ABB RobotStudio station: ABBRoboChallenge2022.rspag

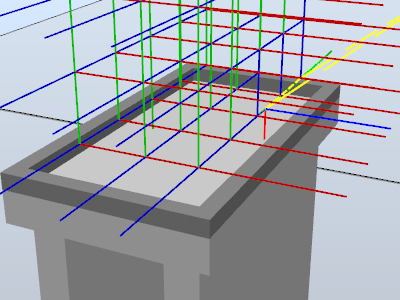
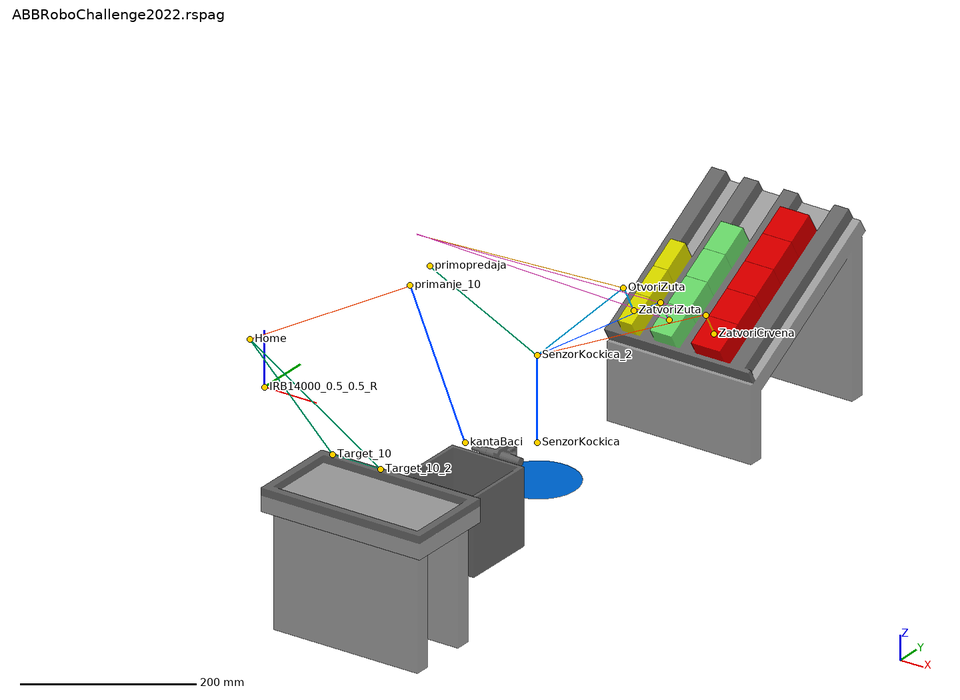
[picture v1: parts stored in the station drawn from their meshes, with robot base, taught points and paths (robot models come from the ABB library and are not in the file)]
--- station ---
Station Solution3 (saved by RobotStudio 22.3.10098.0)
Controller IRB14000, task T_ROB_L: task frame (RAPID world) sits at (0, 0, 100) mm in the station
Controller IRB14000, task T_ROB_R: task frame (RAPID world) sits at (0, 0, 100) mm in the station
Controller IRB14000
  mechanical unit ROB_R: IRB14000_0.5_0.5_R, 6 joints, base frame (0, 0, 0) mm
  mechanical unit ROB_R_7: IRB14000_0.5_0.5_R, 1 joints, base frame (0, 0, 0) mm
  mechanical unit ROB_L: IRB14000_0.5_0.5_L, 6 joints, base frame (0, 0, 0) mm
  mechanical unit ROB_L_7: IRB14000_0.5_0.5_L, 1 joints, base frame (0, 0, 0) mm
Layout (positions relative to the parent item):
  - IRB14000_0.5_0.5 [mechanism, from Robots\IRB14000_0.5_0.5__01.rslib] at (0, 0, 100) mm
  - IRB14000_0.5_0.5_R [mechanism, from Robots\IRB14000_0.5_0.5__01.rslib] at (0, 0, 100) mm; joint values [0.9031, -2.4871, -1.4074, 0.8318, -1.2822, 1.4209, -0.1871] (rad or m)
  - IRB14000_0.5_0.5_L [mechanism, from Robots\IRB14000_0.5_0.5__01.rslib] at (0, 0, 100) mm; joint values [-0.8577, -2.4871, 1.5284, 0.8395, 1.3372, 1.3689, -1.3488] (rad or m)
  - Smart_Gripper_Servo_One_Vacuum_Fingers [mechanism, from Tools\ABB_Smart_Gripper_Servo_One_Vacuum_Fingers.rslib] at (215.12, 134.2, 304.86) mm, rotated rx 113.54 ry -90 rz -23.54 deg; joint values [0] (rad or m)
  - Smart_Gripper_Servo_One_Vacuum_Camera_Fingers [mechanism, from Tools\ABB_Smart_Gripper_Servo_One_Vacuum_Camera_Fingers.rslib] at (228.58, -152.41, 307.36) mm, rotated rx 90 ry 0 rz -180 deg; joint values [0] (rad or m)
  - Senzor_Metala [part] at (250, 150, 15) mm, rotated rx 0 ry 0 rz 180 deg, size 65 x 32 x 27 mm
  - Mesto za testiranje [part] at (275, 150, 0) mm, size 100 x 99.5 x 0 mm
  - Rampa sa kutijama [graphiccomponentgroup]
    - Part_20 [part] at (374.5, 471.2, 184.6) mm, rotated rx 30 ry 0 rz 0 deg, size 40 x 40 x 40 mm
    - Part_1 [part] at (250, 320, 0) mm, size 200 x 20 x 100 mm
    - Part_2 [part] at (250, 520, 0) mm, size 200 x 20 x 200 mm
    - Part_3 [part], size 200 x 226.5 x 142.3 mm
    - Part_4 [part], size 200 x 14.3 x 19.8 mm
    - Part_5 [part], size 20 x 217.8 x 137.3 mm
    - Part_6 [part] at (45, 0, 0) mm, size 20 x 217.8 x 137.3 mm
    - Part_7 [part] at (100, 0, 0) mm, size 20 x 217.8 x 137.3 mm
    - Part_8 [part] at (170, 0, 0) mm, size 20 x 217.8 x 137.3 mm
    - Part_9 [part] at (292.5, 329.17, 102.6) mm, rotated rx 30 ry 0 rz 0 deg, size 20 x 40 x 40 mm
    - Part_10 [part] at (292.5, 364.68, 123.1) mm, rotated rx 30 ry 0 rz 0 deg, size 20 x 40 x 40 mm
    - Part_11 [part] at (292.5, 400.18, 143.6) mm, rotated rx 30 ry 0 rz 0 deg, size 20 x 40 x 40 mm
    - Part_12 [part] at (317.5, 329.17, 102.6) mm, rotated rx 30 ry 0 rz 0 deg, size 30 x 40 x 40 mm
    - Part_13 [part] at (317.5, 364.68, 123.1) mm, rotated rx 30 ry 0 rz 0 deg, size 30 x 40 x 40 mm
    - Part_14 [part] at (317.5, 400.18, 143.6) mm, rotated rx 30 ry 0 rz 0 deg, size 30 x 40 x 40 mm
    - Part_15 [part] at (374.5, 329.17, 102.6) mm, rotated rx 30 ry 0 rz 0 deg, size 40 x 40 x 40 mm
    - Part_16 [part] at (374.5, 364.68, 123.1) mm, rotated rx 30 ry 0 rz 0 deg, size 40 x 40 x 40 mm
    - Part_17 [part] at (374.5, 400.18, 143.6) mm, rotated rx 30 ry 0 rz 0 deg, size 40 x 40 x 40 mm
    - Part_18 [part] at (317.5, 435.69, 164.1) mm, rotated rx 30 ry 0 rz 0 deg, size 30 x 40 x 40 mm
    - Part_19 [part] at (374.5, 435.69, 164.1) mm, rotated rx 30 ry 0 rz 0 deg, size 40 x 40 x 40 mm
  - Paleta [graphiccomponentgroup]
    - Part_31 [part] at (450, -340, 170) mm, size 10 x 100 x 10 mm
    - Part_21 [part] at (250, -340, 0) mm, size 200 x 20 x 150 mm
    - Part_22 [part] at (250, -260, 0) mm, size 200 x 20 x 150 mm
    - Part_25 [part] at (240, -350, 170) mm, size 220 x 10 x 10 mm
    - Part_26 [part] at (240, -240, 170) mm, size 220 x 10 x 10 mm
    - Part_27 [part] at (240, -350, 150) mm, size 220 x 120 x 20 mm
    - Part_28 [part] at (240, -340, 170) mm, size 10 x 100 x 10 mm
  - Mesto za odlaganje [part], size 100 x 100 x 100 mm
Attachment: Smart_Gripper_Servo_One_Vacuum_Fingers is attached to IRB14000_0.5_0.5_L / Link7
Attachment: Smart_Gripper_Servo_One_Vacuum_Camera_Fingers is attached to IRB14000_0.5_0.5_R / Link7
Attachment: Part_8 is attached to Part_7
Attachment: Part_7 is attached to Part_6
Attachment: Part_6 is attached to Part_5
Attachment: Part_5 is attached to Part_4
Attachment: Part_4 is attached to Part_3
Attachment: Part_3 is attached to Part_2
Attachment: Part_2 is attached to Part_1
Attachment: Part_9 is attached to Part_4
Attachment: Part_10 is attached to Part_4
Attachment: Part_11 is attached to Part_4
Attachment: Part_12 is attached to Part_4
Attachment: Part_13 is attached to Part_4
Attachment: Part_14 is attached to Part_4
Attachment: Part_15 is attached to Part_4
Attachment: Part_16 is attached to Part_4
Attachment: Part_17 is attached to Part_4
Attachment: Part_18 is attached to Part_4
Attachment: Part_19 is attached to Part_4
Attachment: Part_20 is attached to Part_4
Attachment: Part_31 is attached to Part_28
Attachment: Part_28 is attached to Part_26
Attachment: Part_26 is attached to Part_25
Attachment: Part_25 is attached to Part_27
Attachment: Part_27 is attached to Part_22
Attachment: Part_22 is attached to Part_21
Targets, tools, work objects and paths stored in the station and not in the controller backup, written as RAPID:
! task T_ROB_L
MODULE Module1
  CONST robtarget SenzorKockica_2_4:=[[0,0,-0.911663764],[0,-0.707106781,0.707106781,0],[-1,0,1,5],[103.674755702,9E+09,9E+09,9E+09,9E+09,9E+09]];
  CONST robtarget SenzorKockica_4:=[[0,0,128.036682994],[0,0.707106781,0.707106781,0],[-1,0,1,5],[103.674755702,9E+09,9E+09,9E+09,9E+09,9E+09]];
ENDMODULE


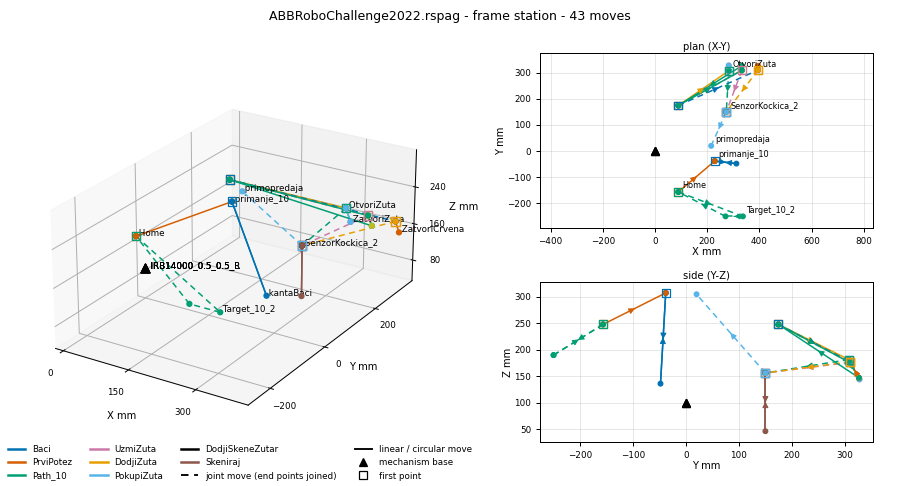
[picture p0: tool path of ABBRoboChallenge2022.rspag in frame station, 43 of 43 moves have a stored position in this frame; points joined in program order, loops and branches not executed]
--- Backups/IRB14000/RAPID/TASK1/PROGMOD/CalibData.mod ---
MODULE CalibData
    PERS tooldata Servo:=[TRUE,[[0,0,114.2],[1,0,0,0]],[0.24,[8.2,12.5,48.1],[1,0,0,0],0.00022,0.00024,0.00009]];
    PERS tooldata VaccumOne:=[TRUE,[[63.5,18.5,37.5],[0.707106781,0,0.707106781,0]],[0.24,[8.2,12.5,48.1],[1,0,0,0],0.00022,0.00024,0.00009]];
    PERS tooldata Camera:=[TRUE,[[-7.3,28.3,35.1],[0.5,-0.5,0.5,0.5]],[0.24,[8.2,12.5,48.1],[1,0,0,0],0.00022,0.00024,0.00009]];
    PERS wobjdata Workobject_2:=[FALSE,TRUE,"",[[311.493,-47.839,34.371],[1,0,0,0]],[[0,0,0],[1,0,0,0]]];
   PERS wobjdata Workobject_3:=[FALSE,TRUE,"",[[270,-250,90],[0.5,0.5,0.5,0.5]],[[0,0,0],[0.707106781,-0.707106781,0,0]]];
    PERS wobjdata Workobject_4:=[FALSE,TRUE,"",[[310,-250,90],[0.5,0.5,0.5,0.5]],[[0,0,0],[0.707106781,-0.707106781,0,0]]];
    PERS wobjdata Workobject_5:=[FALSE,TRUE,"",[[350,-250,90],[0.5,0.5,0.5,0.5]],[[0,0,0],[0.707106781,-0.707106781,0,0]]];
    PERS wobjdata Workobject_6:=[FALSE,TRUE,"",[[390,-250,90],[0.5,0.5,0.5,0.5]],[[0,0,0],[1,0,0,0]]];
    PERS wobjdata Workobject_7:=[FALSE,TRUE,"",[[430,-250,90],[0.5,0.5,0.5,0.5]],[[0,0,0],[1,0,0,0]]];
    PERS wobjdata Workobject_8:=[FALSE,TRUE,"",[[430,-320,90],[0.5,0.5,0.5,0.5]],[[0,0,0],[1,0,0,0]]];
    PERS wobjdata Workobject_9:=[FALSE,TRUE,"",[[390,-320,90],[0.5,0.5,0.5,0.5]],[[0,0,0],[1,0,0,0]]];
    PERS wobjdata Workobject_10:=[FALSE,TRUE,"",[[390,-280,90],[0.5,0.5,0.5,0.5]],[[0,0,0],[1,0,0,0]]];
    PERS wobjdata Workobject_11:=[FALSE,TRUE,"",[[430,-280,90],[0.5,0.5,0.5,0.5]],[[0,0,0],[1,0,0,0]]];
    PERS wobjdata Workobject_12:=[FALSE,TRUE,"",[[270,-320,90],[0.5,0.5,0.5,0.5]],[[0,0,0],[1,0,0,0]]];
    PERS wobjdata Workobject_13:=[FALSE,TRUE,"",[[270,-280,90],[0.5,0.5,0.5,0.5]],[[0,0,0],[1,0,0,0]]];
    PERS wobjdata Workobject_14:=[FALSE,TRUE,"",[[310,-320,90],[0.5,0.5,0.5,0.5]],[[0,0,0],[1,0,0,0]]];
    PERS wobjdata Workobject_15:=[FALSE,TRUE,"",[[310,-280,90],[0.5,0.5,0.5,0.5]],[[0,0,0],[1,0,0,0]]];
    PERS wobjdata Workobject_16:=[FALSE,TRUE,"",[[350,-280,90],[0.5,0.5,0.5,0.5]],[[0,0,0],[1,0,0,0]]];
    PERS wobjdata Workobject_17:=[FALSE,TRUE,"",[[350,-320,90],[0.5,0.5,0.5,0.5]],[[0,0,0],[0,1,0,0]]];
    PERS wobjdata Workobject_21:=[FALSE,TRUE,"",[[430,-320,130],[0.5,0.5,0.5,0.5]],[[0,0,0],[1,0,0,0]]];
    PERS wobjdata Workobject_22:=[FALSE,TRUE,"",[[390,-320,130],[0.5,0.5,0.5,0.5]],[[0,0,0],[1,0,0,0]]];
    PERS wobjdata Workobject_23:=[FALSE,TRUE,"",[[350,-320,130],[0.5,0.5,0.5,0.5]],[[0,0,0],[1,0,0,0]]];
    PERS wobjdata Workobject_24:=[FALSE,TRUE,"",[[310,-320,130],[0.5,0.5,0.5,0.5]],[[0,0,0],[1,0,0,0]]];
    PERS wobjdata Workobject_25:=[FALSE,TRUE,"",[[270,-320,130],[0.5,0.5,0.5,0.5]],[[0,0,0],[1,0,0,0]]];
    PERS wobjdata Workobject_26:=[FALSE,TRUE,"",[[270,-280,130],[0.5,0.5,0.5,0.5]],[[0,0,0],[1,0,0,0]]];
    PERS wobjdata Workobject_27:=[FALSE,TRUE,"",[[310,-280,130],[0.5,0.5,0.5,0.5]],[[0,0,0],[1,0,0,0]]];
    PERS wobjdata Workobject_28:=[FALSE,TRUE,"",[[350,-280,130],[0.5,0.5,0.5,0.5]],[[0,0,0],[1,0,0,0]]];
    PERS wobjdata Workobject_29:=[FALSE,TRUE,"",[[390,-280,130],[0.5,0.5,0.5,0.5]],[[0,0,0],[1,0,0,0]]];
    PERS wobjdata Workobject_30:=[FALSE,TRUE,"",[[430,-280,130],[0.5,0.5,0.5,0.5]],[[0,0,0],[1,0,0,0]]];
    PERS wobjdata Workobject_31:=[FALSE,TRUE,"",[[270,-250,130],[0.5,0.5,0.5,0.5]],[[0,0,0],[1,0,0,0]]];
    PERS wobjdata Workobject_32:=[FALSE,TRUE,"",[[310,-250,130],[0.5,0.5,0.5,0.5]],[[0,0,0],[1,0,0,0]]];
    PERS wobjdata Workobject_33:=[FALSE,TRUE,"",[[350,-250,130],[0.5,0.5,0.5,0.5]],[[0,0,0],[1,0,0,0]]];
    PERS wobjdata Workobject_34:=[FALSE,TRUE,"",[[390,-250,130],[0.5,0.5,0.5,0.5]],[[0,0,0],[1,0,0,0]]];
    PERS wobjdata Workobject_35:=[FALSE,TRUE,"",[[430,-250,130],[0.5,0.5,0.5,0.5]],[[0,0,0],[1,0,0,0]]];
    PERS wobjdata Workobject_36:=[FALSE,TRUE,"",[[430,-320,170],[0.5,0.5,0.5,0.5]],[[0,0,0],[1,0,0,0]]];
    PERS wobjdata Workobject_37:=[FALSE,TRUE,"",[[270,-320,170],[0.5,0.5,0.5,0.5]],[[0,0,0],[1,0,0,0]]];
    PERS wobjdata Workobject_38:=[FALSE,TRUE,"",[[270,-280,170],[0.5,0.5,0.5,0.5]],[[0,0,0],[1,0,0,0]]];
    PERS wobjdata Workobject_39:=[FALSE,TRUE,"",[[310,-320,170],[0.5,0.5,0.5,0.5]],[[0,0,0],[1,0,0,0]]];
    PERS wobjdata Workobject_40:=[FALSE,TRUE,"",[[310,-280,170],[0.5,0.5,0.5,0.5]],[[0,0,0],[1,0,0,0]]];
    PERS wobjdata Workobject_41:=[FALSE,TRUE,"",[[270,-250,170],[0.5,0.5,0.5,0.5]],[[0,0,0],[1,0,0,0]]];
    PERS wobjdata Workobject_42:=[FALSE,TRUE,"",[[310,-250,170],[0.5,0.5,0.5,0.5]],[[0,0,0],[1,0,0,0]]];
    PERS wobjdata Workobject_43:=[FALSE,TRUE,"",[[350,-320,170],[0.5,0.5,0.5,0.5]],[[0,0,0],[1,0,0,0]]];
    PERS wobjdata Workobject_44:=[FALSE,TRUE,"",[[350,-280,170],[0.5,0.5,0.5,0.5]],[[0,0,0],[1,0,0,0]]];
    PERS wobjdata Workobject_45:=[FALSE,TRUE,"",[[350,-250,170],[0.5,0.5,0.5,0.5]],[[0,0,0],[1,0,0,0]]];
    PERS wobjdata Workobject_46:=[FALSE,TRUE,"",[[390,-320,170],[0.5,0.5,0.5,0.5]],[[0,0,0],[1,0,0,0]]];
    PERS wobjdata Workobject_47:=[FALSE,TRUE,"",[[390,-280,170],[0.5,0.5,0.5,0.5]],[[0,0,0],[1,0,0,0]]];
    PERS wobjdata Workobject_48:=[FALSE,TRUE,"",[[430,-250,170],[0.5,0.5,0.5,0.5]],[[0,0,0],[1,0,0,0]]];
    PERS wobjdata Workobject_49:=[FALSE,TRUE,"",[[390,-250,170],[0.5,0.5,0.5,0.5]],[[0,0,0],[1,0,0,0]]];
    PERS wobjdata Workobject_50:=[FALSE,TRUE,"",[[430,-280,170],[0.5,0.5,0.5,0.5]],[[0,0,0],[1,0,0,0]]];
    PERS wobjdata Workobject_51:=[FALSE,TRUE,"",[[265,-20,190],[1,0,0,0]],[[0,0,0],[1,0,0,0]]];
    PERS wobjdata Kanta:=[FALSE,TRUE,"",[[311.493,-47.839,34.371],[0,1,0,0]],[[0,0,0],[1,0,0,0]]];
    PERS wobjdata Primanje:=[FALSE,TRUE,"",[[265,-20,190],[1,0,0,0]],[[0,0,0],[1,0,0,0]]];
    PERS wobjdata Workobject_1:=[FALSE,TRUE,"",[[273,150,-53.701],[1,0,0,0]],[[0,0,0],[1,0,0,0]]];
    PERS wobjdata KockicaZ:=[FALSE,TRUE,"",[[282.5,326.49,47.239],[0.969411434,0.245441382,0,0]],[[0,0,0],[1,0,0,0]]];
    PERS wobjdata Workobject_19:=[FALSE,TRUE,"",[[332.5,326.491,47.241],[1,0,0,0]],[[0,0,0],[1,0,0,0]]];
    PERS wobjdata Workobject_20:=[FALSE,TRUE,"",[[394.5,326.491,47.241],[0.608400247,-0.360345861,0.608400247,-0.360345861]],[[0,0,0],[1,0,0,0]]];
    PERS wobjdata Workobject_53:=[FALSE,TRUE,"",[[265,-26.752845654,190],[0.5,0.5,0.5,0.5]],[[0,0,0],[1,0,0,0]]];
ENDMODULE

--- Backups/IRB14000/RAPID/TASK1/PROGMOD/Module1.mod ---
MODULE Module1
        CONST robtarget primanje_10:=[[-36.418450574,-18.209391177,17.355412881],[0,0,0.707106781,0.707106781],[1,-1,0,4],[-101.964427132,9E+09,9E+09,9E+09,9E+09,9E+09]];
    CONST robtarget kanta_10:=[[0,0,0],[1,0,0,0],[-1,0,1,1],[-111.964425004,9E+09,9E+09,9E+09,9E+09,9E+09]];
    CONST robtarget Home:=[[89.387946422,-156.622117956,147.913470217],[0.066010726,-0.842420918,-0.111214912,-0.523068661],[0,0,0,4],[-101.964427132,9E+09,9E+09,9E+09,9E+09,9E+09]];
    CONST robtarget primopredaja_2:=[[0,0,0],[0.5,0.5,-0.5,0.5],[1,0,2,1],[103.674760418,9E+09,9E+09,9E+09,9E+09,9E+09]];
    CONST robtarget primanje_10_2:=[[0.267352692,0.235735351,-1.691583869],[0,0,0,1],[1,-1,0,4],[-101.964427132,9E+09,9E+09,9E+09,9E+09,9E+09]];
    CONST robtarget kantaBaci:=[[0.267352692,0.235735351,-1.691583869],[0,0,0,1],[1,-1,0,4],[-101.964427132,9E+09,9E+09,9E+09,9E+09,9E+09]];
    CONST robtarget Target_10:=[[0,0,0],[1,0,0,0],[1,0,-1,5],[-101.964427132,9E+09,9E+09,9E+09,9E+09,9E+09]];
    CONST robtarget Target_10_2:=[[0,-66.608628748,0],[0.707106781,0,0.707106781,0],[1,0,-1,5],[-101.964427132,9E+09,9E+09,9E+09,9E+09,9E+09]];
    CONST robtarget Target_20:=[[0,0,0],[1,0,0,0],[0,0,0,0],[-101.964417119,9E+09,9E+09,9E+09,9E+09,9E+09]];
    PROC main()
        Path_10;
    ENDPROC
    PROC Baci()
        MoveL primanje_10,v1000,z100,Servo\WObj:=Primanje;
        MoveL kantaBaci,v1000,z100,Servo\WObj:=Kanta;
        MoveL primanje_10,v1000,z100,Servo\WObj:=Primanje;
    ENDPROC
    PROC PrviPotez()
        MoveL Home,v1000,z100,Servo\WObj:=wobj0;
        MoveL primanje_10,v1000,z100,Servo\WObj:=Primanje;
    ENDPROC
    PROC Path_10()
        MoveL Home,v1000,z100,Servo\WObj:=wobj0;
        MoveJ Target_10_2,v1000,z100,Servo\WObj:=Workobject_3;
        MoveJ Target_10,v1000,z100,Servo\WObj:=Workobject_3;
        MoveJ Home,v1000,z100,Servo\WObj:=wobj0;
    ENDPROC
ENDMODULE

--- Backups/IRB14000/RAPID/TASK2/PROGMOD/CalibData.mod ---
MODULE CalibData
    PERS tooldata Servo:=[TRUE,[[0,0,114.2],[1,0,0,0]],[0.226,[8.9,12.3,48.7],[1,0,0,0],0.00021,0.00024,0.00009]];
    PERS tooldata VaccumOne:=[TRUE,[[63.5,18.5,37.5],[0.707106781,0,0.707106781,0]],[0.226,[8.9,12.3,48.7],[1,0,0,0],0.00021,0.00024,0.00009]];
    PERS wobjdata Workobject_1:=[FALSE,TRUE,"",[[273,150,-53.701],[1,0,0,0]],[[0,0,0],[1,0,0,0]]];
    PERS wobjdata KockicaZ:=[FALSE,TRUE,"",[[282.5,326.49,47.239],[0.969411434,0.245441382,0,0]],[[0,0,0],[1,0,0,0]]];
    PERS wobjdata Workobject_19:=[FALSE,TRUE,"",[[332.5,326.491,47.241],[1,0,0,0]],[[0,0,0],[1,0,0,0]]];
    PERS wobjdata Workobject_20:=[FALSE,TRUE,"",[[394.5,326.491,47.241],[0.248054386,-0.968746108,0,0]],[[0,0,0],[1,0,0,0]]];
    PERS wobjdata Workobject_51:=[FALSE,TRUE,"",[[265,-20,190],[1,0,0,0]],[[0,0,0],[1,0,0,0]]];
    PERS wobjdata Workobject_53:=[FALSE,TRUE,"",[[265,20,190],[1,0,0,0]],[[0,0,0],[1,0,0,0]]];
ENDMODULE

--- Backups/IRB14000/RAPID/TASK2/PROGMOD/Module1.mod ---
MODULE Module1
    CONST robtarget Home:=[[89.388081176,174.575150508,147.913525533],[0.06601065,0.842420935,-0.111215019,0.52306862],[0,0,0,4],[101.964427489,9E+09,9E+09,9E+09,9E+09,9E+09]];
    CONST robtarget OtvoriZuta:=[[0,-0.475935817,39.28134243],[-0.000001405,1,0,0],[-1,-2,2,4],[101.964427132,9E+09,9E+09,9E+09,9E+09,9E+09]];
    CONST robtarget ZatvoriZuta:=[[0,-0.476055148,-3.185077172],[-0.000001405,1,0,0],[-1,-2,2,4],[101.964427132,9E+09,9E+09,9E+09,9E+09,9E+09]];
    CONST robtarget SenzorKockica_2:=[[0,0,109.884559664],[0,-0.707106781,0.707106781,0],[-1,0,1,5],[103.674755702,9E+09,9E+09,9E+09,9E+09,9E+09]];
    CONST robtarget SenzorKockica:=[[0,0,0],[0,0.707106781,0.707106781,0],[-1,0,1,5],[103.674755702,9E+09,9E+09,9E+09,9E+09,9E+09]];
    CONST robtarget primopredaja:=[[-49.881892864,0,14.861905631],[0.5,0.5,-0.5,0.5],[-1,1,-1,4],[103.674760418,9E+09,9E+09,9E+09,9E+09,9E+09]];
    CONST robtarget OtvoriZelena:=[[0,-17.44947162,28.955893491],[0.267861537,-0.963457418,0,0],[-1,-2,2,4],[103.674755702,9E+09,9E+09,9E+09,9E+09,9E+09]];
    CONST robtarget ZatvoriZelena:=[[0,0,0],[0.267861537,-0.963457418,0,0],[-1,-2,2,4],[103.674755702,9E+09,9E+09,9E+09,9E+09,9E+09]];
    CONST robtarget OtvoriCrvena:=[[0,0,-34.27342111],[1,0,0,0],[-1,-2,-2,4],[103.674755702,9E+09,9E+09,9E+09,9E+09,9E+09]];
    CONST robtarget ZatvoriCrvena:=[[0,0,0],[1,0,0,0],[-1,-2,-2,4],[103.674755702,9E+09,9E+09,9E+09,9E+09,9E+09]];
    CONST robtarget SenzorKockica_gore_2:=[[0,0,109.884559664],[0,0,1,0],[-1,0,2,5],[103.674755702,9E+09,9E+09,9E+09,9E+09,9E+09]];
    CONST robtarget SenzorKockica_dole_3:=[[0,0,0],[0,0,1,0],[-1,0,2,5],[103.674755702,9E+09,9E+09,9E+09,9E+09,9E+09]];


    PERS tasks task_list{2}:=[["T_ROB_L"], ["T_ROB_R"]];
    VAR syncident sync1;
    VAR syncident sync2;
    VAR num sum:=0;
    VAR num k1:=-1;
    VAR num k3:=-1;
    VAR num k2:=-1;
    VAR num X;


    PROC UzmiZuta()
        MoveL OtvoriZuta,v100,fine,Servo\WObj:=KockicaZ;
        MoveL ZatvoriZuta,v100,fine,Servo\WObj:=KockicaZ;
        MoveJ OtvoriZuta,v100,fine,Servo\WObj:=KockicaZ;


    ENDPROC


    PROC DodjiZuta()
        MoveL Home,v500,fine,Servo\WObj:=wobj0;
        MoveL OtvoriZuta,v500,fine,Servo\WObj:=KockicaZ;
    ENDPROC
    PROC PokupiZuta()
        MoveL OtvoriZuta,v100,fine,Servo\WObj:=KockicaZ;
        MoveL ZatvoriZuta,v100,fine,Servo\WObj:=KockicaZ;
        MoveL OtvoriZuta,v100,fine,Servo\WObj:=KockicaZ;
    ENDPROC
    PROC DodjiSkeneZutar()
        MoveL SenzorKockica_2,v500,fine,Servo\WObj:=Workobject_1;
    ENDPROC
    PROC Skeniraj()
        MoveL SenzorKockica_2,v500,fine,Servo\WObj:=Workobject_1;
        MoveL SenzorKockica,v500,fine,Servo\WObj:=Workobject_1;
        MoveL SenzorKockica_2,v500,fine,Servo\WObj:=Workobject_1;
    ENDPROC
    PROC DodjiZelena()
        MoveJ Home,v500,z100,Servo\WObj:=wobj0;
        MoveJ OtvoriZelena,v500,z100,Servo\WObj:=Workobject_19;
    ENDPROC
    PROC UzmiZelena()
        MoveJ OtvoriZelena,v100,z100,Servo\WObj:=Workobject_19;
        MoveJ ZatvoriZelena,v100,z100,Servo\WObj:=Workobject_19;
        MoveJ OtvoriZelena,v100,z100,Servo\WObj:=Workobject_19;
    ENDPROC
    PROC DodjiCrvena()
        MoveJ Home,v500,z100,Servo\WObj:=wobj0;
        MoveJ OtvoriCrvena,v500,z100,Servo\WObj:=Workobject_20;
    ENDPROC
    PROC UzmiCrvena()
        MoveJ OtvoriCrvena,v100,z100,Servo\WObj:=Workobject_20;
        MoveJ ZatvoriCrvena,v100,z100,Servo\WObj:=Workobject_20;
        MoveJ OtvoriCrvena,v100,z100,Servo\WObj:=Workobject_20;
    ENDPROC
    PROC DodjiSkenerZuta()
        MoveJ OtvoriZuta,v500,z100,Servo\WObj:=KockicaZ;
        MoveJ SenzorKockica_2,v500,z100,Servo\WObj:=Workobject_1;
    ENDPROC
    PROC DodjiSkenerZelena()
        MoveJ OtvoriZelena,v500,z100,Servo\WObj:=Workobject_19;
        MoveJ SenzorKockica_2,v500,z100,Servo\WObj:=Workobject_1;
    ENDPROC
    PROC DodjiSkenerCrvena()
        MoveJ OtvoriCrvena,v500,z100,Servo\WObj:=Workobject_20;
        MoveJ SenzorKockica_2,v500,z100,Servo\WObj:=Workobject_1;
    ENDPROC
    PROC Predaja()
        MoveJ SenzorKockica_2,v500,z100,Servo\WObj:=Workobject_1;
        MoveJ primopredaja,v500,z100,Servo\WObj:=Workobject_53;
    ENDPROC
    PROC Path_10()
        MoveL Home,v1000,z100,Servo\WObj:=wobj0;
        MoveL OtvoriZelena,v1000,z100,Servo\WObj:=Workobject_19;
        MoveL ZatvoriZelena,v1000,z100,Servo\WObj:=Workobject_19;
        MoveL Home,v1000,z100,Servo\WObj:=wobj0;
        DodjiZelena;
    ENDPROC


    PROC main()

        Hand_Initialize \maxSpd:=20, \holdForce:=12;
        Hand_JogOutward;
        TPWrite("Dobro dosli! Unesite opciju za slaganje kockica u paleti");
        TPReadNum X, "1-Jedna boja kockica, 2-Dve boje kockica, 3-3 boje kockica";
            IF X=2 then
                TPReadNum k1, "Unesite prvu boju kockica";
                TPReadNum k2, "Unesite drugu boju kockica";
                sum:=30;

                IF(k1=1 OR k2=1)
                    FOR i FROM 0 TO 15 DO
                    ENDFOR
                 ENDIF


                IF(k1=2 OR k2=2)
                    FOR i FROM 0 TO 15 DO
                        DodjiZelena;
                        UzmiZelena;
                        DodjiSkenerZelena;
                        Skeniraj;
                    ENDFOR


                 IF(k1=3 or k2=3)
                    FOR i FROM 0 TO 15 DO
                    ENDFOR




           ELSEIF(X=1)
                TPReadNum k1, "Unesite prvu boju kockica";
                sum:=15;

                IF(k1=1)
                FOR i FROM 0 TO 15 DO
                        Predaja;
                ENDFOR

                IF(k1=2)
                    FOR i FROM 0 TO 15 DO
                ENDFOR

                 IF(k1=3)
                    FOR i FROM 0 TO 15 DO
                        DodjiCrvena;
                ENDFOR

                ELSEIF (X=3)
                    TPWrite("Izabrane su sve tri boje kockica");
                    k1:=1; k2:=2; k3:=3;

                    FOR i FROM 0 TO 15 DO
                    ENDFOR


                FOR i FROM 0 TO 15 DO
                ENDFOR


                FOR i FROM 0 TO 15 DO
                    UzmiCrvena;
                ENDFOR



             ELSE TPWrite("Upps dozvoljeno je uneti samo neki od brojeva 1, 2 ili 3");






    ENDPROC
ENDMODULE




        DodjiZelena;
        UzmiZelena;
        DodjiSkenerZelena;
        Skeniraj;
        Predaja;
        DodjiCrvena;
        UzmiCrvena;
    ENDPROC

ENDMODULE

--- Backups/IRB14000/SYSPAR/EIO.cfg ---
EIO:CFG_1.0:6:1::
#
SYSSIG_IN:

      -Signal "Collision_Avoidance" -Action "CollAvoidance"
#
INDUSTRIAL_NETWORK:

      -Name "EtherNetIP" -Connection "Private Network" -Label "EtherNet/IP"

      -Name "DeviceNet" -Label "DeviceNet Master/Slave Network" -Address "2"
#
EIO_CROSS:

      -Name "Cross_Signal_Lamp" -Res "Signal_Lamp" -Act1 "DRV1BRAKE"
#
EIO_SIGNAL_SAFELEVEL:

      -Name "FlangePowerSafeLevel" -ActionWhenStartup "Last"

      -Name "SGcmdSafeLevel" -ActionWhenAccessible "Default"
#
ETHERNETIP_DEVICE:

      -Name "Hand_R" -StateWhenStartup "Deactivated" -VendorName "ABB"\
      -ProductName "EtherNet/IP EIP" -Label "2" -Address "192.168.125.30"\
      -VendorId 75 -ProductCode 1 -OutputAssembly 100 -InputAssembly 101\
      -InputConnectionType "POINT2POINT" -OutputSize 10 -InputSize 10\
      -O2T_RPI 10000 -T2O_RPI 10000 -ConnectionTimeoutMultiplier 2

      -Name "Hand_L" -StateWhenStartup "Deactivated" -VendorName "ABB"\
      -ProductName "EtherNet/IP EIP" -Label "1" -Address "192.168.125.40"\
      -VendorId 75 -ProductCode 1 -OutputAssembly 100 -InputAssembly 101\
      -InputConnectionType "POINT2POINT" -OutputSize 10 -InputSize 10\
      -O2T_RPI 10000 -T2O_RPI 10000 -ConnectionTimeoutMultiplier 2
#
DEVICENET_DEVICE:

      -Name "D652_10" -VendorName "ABB Robotics" -ProductName "24 VDC Unit"\
      -Address 10 -ProductCode 26 -DeviceType 7 -ConnectionType "COS"\
      -OutputSize 2 -InputSize 2
#
DEVICENET_INTERNAL_DEVICE:

      -Name "DN_Internal_Device" -VendorName "ABB Robotics"\
      -ProductName "DeviceNet Internal Slave Device"
#
ETHERNETIP_INTERNAL_DEVICE:

      -Name "EN_Internal_Device" -VendorName "ABB Robotics"\
      -ProductName "EtherNet/IP Internal Adapter Device"
#
EIO_SIGNAL:

      -Name "custom_DI_0" -SignalType "DI" -Device "D652_10" -DeviceMap "0"

      -Name "custom_DI_1" -SignalType "DI" -Device "D652_10" -DeviceMap "1"

      -Name "custom_DI_2" -SignalType "DI" -Device "D652_10" -DeviceMap "2"

      -Name "custom_DI_3" -SignalType "DI" -Device "D652_10" -DeviceMap "3"

      -Name "custom_DI_4" -SignalType "DI" -Device "D652_10" -DeviceMap "4"

      -Name "custom_DI_5" -SignalType "DI" -Device "D652_10" -DeviceMap "5"

      -Name "custom_DI_6" -SignalType "DI" -Device "D652_10" -DeviceMap "6"

      -Name "custom_DI_7" -SignalType "DI" -Device "D652_10" -DeviceMap "7"

      -Name "custom_DO_0" -SignalType "DO" -Device "D652_10" -DeviceMap "0"

      -Name "custom_DO_1" -SignalType "DO" -Device "D652_10" -DeviceMap "1"

      -Name "custom_DO_2" -SignalType "DO" -Device "D652_10" -DeviceMap "2"

      -Name "custom_DO_3" -SignalType "DO" -Device "D652_10" -DeviceMap "3"

      -Name "custom_DO_4" -SignalType "DO" -Device "D652_10" -DeviceMap "4"

      -Name "custom_DO_5" -SignalType "DO" -Device "D652_10" -DeviceMap "5"

      -Name "custom_DO_6" -SignalType "DO" -Device "D652_10" -DeviceMap "6"

      -Name "custom_DO_7" -SignalType "DO" -Device "D652_10" -DeviceMap "7"

      -Name "hall_sensor_joint_1" -SignalType "DI" -Device "D652_10"\
      -DeviceMap "8"

      -Name "hall_sensor_joint_2" -SignalType "DI" -Device "D652_10"\
      -DeviceMap "9"

      -Name "hall_sensor_joint_3" -SignalType "DI" -Device "D652_10"\
      -DeviceMap "11"

      -Name "hall_sensor_joint_4" -SignalType "DI" -Device "D652_10"\
      -DeviceMap "12"

      -Name "hall_sensor_joint_5" -SignalType "DI" -Device "D652_10"\
      -DeviceMap "13"

      -Name "hall_sensor_joint_6" -SignalType "DI" -Device "D652_10"\
      -DeviceMap "14"

      -Name "hall_sensor_joint_7" -SignalType "DI" -Device "D652_10"\
      -DeviceMap "10"

      -Name "hall_sensor_24V_ROB_R" -SignalType "DO" -Device "D652_10"\
      -DeviceMap "8"

      -Name "hall_sensor_24V_ROB_L" -SignalType "DO" -Device "D652_10"\
      -DeviceMap "9"

      -Name "flange_24V_ROB_R" -SignalType "DO" -Device "D652_10"\
      -DeviceMap "10" -SafeLevel "FlangePowerSafeLevel"

      -Name "flange_24V_ROB_L" -SignalType "DO" -Device "D652_10"\
      -DeviceMap "11" -SafeLevel "FlangePowerSafeLevel"

      -Name "Signal_Lamp" -SignalType "DO" -Device "D652_10" -DeviceMap "12"

      -Name "Collision_Avoidance" -SignalType "DO" -Access "All" -Default 1

      -Name "hand_CmdGripper_R" -SignalType "GO" -Device "Hand_R"\
      -Label "Hand Command Right" -DeviceMap "0-4" -Category "HandRight"\
      -Access "All" -SafeLevel "SGcmdSafeLevel"

      -Name "hand_CmdClearErr_R" -SignalType "DO" -Device "Hand_R"\
      -Label "Clear Error Right" -DeviceMap "7" -Category "HandRight"\
      -Access "All"

      -Name "hand_MaxPosition_R" -SignalType "GO" -Device "Hand_R"\
      -Label "Max Position Right" -DeviceMap "8-15" -Category "HandRight"\
      -Access "All" -Default 100

      -Name "hand_MinPosition_R" -SignalType "GO" -Device "Hand_R"\
      -Label "Min Position Right" -DeviceMap "16-23" -Category "HandRight"\
      -Access "All" -Default 50

      -Name "hand_MaxSpeed_R" -SignalType "GO" -Device "Hand_R"\
      -Label "Max Speed Right" -DeviceMap "24-31" -Category "HandRight"\
      -Access "All" -Default 200

      -Name "hand_HoldForce_R" -SignalType "GO" -Device "Hand_R"\
      -Label "Hold Force Right" -DeviceMap "40-47" -Category "HandRight"\
      -Access "All" -Default 120

      -Name "hand_CmdVacuum1_R" -SignalType "DO" -Device "Hand_R"\
      -Label "Vacuum 1 Right" -DeviceMap "48" -Category "HandRight"\
      -Access "All"

      -Name "hand_CmdVacuum2_R" -SignalType "DO" -Device "Hand_R"\
      -Label "Vacuum 2 Right" -DeviceMap "49" -Category "HandRight"\
      -Access "All"

      -Name "hand_CmdBlowoff1_R" -SignalType "DO" -Device "Hand_R"\
      -Label "BlowOff 1 Right" -DeviceMap "50" -Category "HandRight"\
      -Access "All"

      -Name "hand_CmdBlowoff2_R" -SignalType "DO" -Device "Hand_R"\
      -Label "BlowOff 2 Right" -DeviceMap "51" -Category "HandRight"\
      -Access "All"

      -Name "hand_SysState_R" -SignalType "GI" -Device "Hand_R"\
      -Label "Finger State Right" -DeviceMap "0-4" -Category "HandRight"\
      -Access "All"

      -Name "hand_SysError_R" -SignalType "GI" -Device "Hand_R"\
      -Label "Finger Error Right" -DeviceMap "32-39" -Category "HandRight"\
      -Access "All"

      -Name "hand_StatusCalibrated_R" -SignalType "DI" -Device "Hand_R"\
      -Label "Calibrated Right" -DeviceMap "5" -Category "HandRight"\
      -Access "All"

      -Name "hand_ActualPosition_R" -SignalType "GI" -Device "Hand_R"\
      -Label "Actual Position Right" -DeviceMap "8-15" -Category "HandRight"\
      -Access "All"

      -Name "hand_ActualSpeed_R" -SignalType "GI" -Device "Hand_R"\
      -Label "Actual Speed Right" -DeviceMap "16-23" -Category "HandRight"\
      -Access "All"

      -Name "hand_StatusCamLinked_R" -SignalType "DI" -Device "Hand_R"\
      -Label "Camera Connection Right" -DeviceMap "40" -Category "HandRight"\
      -Access "All"

      -Name "hand_SoftwareVersion_R" -SignalType "GI" -Device "Hand_R"\
      -Label "Software Version Right" -DeviceMap "41-47" -Category "HandRight"\
      -Access "All"

      -Name "hand_StatusVacuum1_R" -SignalType "DI" -Device "Hand_R"\
      -Label "Vacuum 1 Right Status" -DeviceMap "48" -Category "HandRight"\
      -Access "All"

      -Name "hand_StatusVacuum2_R" -SignalType "DI" -Device "Hand_R"\
      -Label "Vacuum 1 Right Status" -DeviceMap "49" -Category "HandRight"\
      -Access "All"

      -Name "hand_StatusBlowoff1_R" -SignalType "DI" -Device "Hand_R"\
      -Label "SuncTool 1 Right Status" -DeviceMap "50" -Category "HandRight"\
      -Access "All"

      -Name "hand_StatusBlowoff2_R" -SignalType "DI" -Device "Hand_R"\
      -Label "SuncTool 1 Right Status" -DeviceMap "51" -Category "HandRight"\
      -Access "All"

      -Name "hand_ActualPressure1_R" -SignalType "GI" -Device "Hand_R"\
      -Label "Vacuum pressure1 Right" -DeviceMap "64-71" -Category "HandRight"\
      -Access "All"

      -Name "hand_ActualPressure2_R" -SignalType "GI" -Device "Hand_R"\
      -Label "Vacuum pressure2 Right" -DeviceMap "72-79" -Category "HandRight"\
      -Access "All"

      -Name "hand_SecurityKey_R" -SignalType "GO" -Device "Hand_R"\
      -Label "Security key right" -DeviceMap "64-71" -Category "HandRight"\
      -Access "All"

      -Name "hand_TftPFtpMode_R" -SignalType "DI" -Device "Hand_R"\
      -Label "Hand firmware update mode" -DeviceMap "7" -Category "HandRight"\
      -Access "All"

      -Name "hand_CmdGripper_L" -SignalType "GO" -Device "Hand_L"\
      -Label "Hand Command Left" -DeviceMap "0-4" -Category "HandLeft"\
      -Access "All" -SafeLevel "SGcmdSafeLevel"

      -Name "hand_CmdClearErr_L" -SignalType "DO" -Device "Hand_L"\
      -Label "Clear Error Left" -DeviceMap "7" -Category "HandLeft"\
      -Access "All"

      -Name "hand_MaxPosition_L" -SignalType "GO" -Device "Hand_L"\
      -Label "Max Position Left" -DeviceMap "8-15" -Category "HandLeft"\
      -Access "All" -Default 100

      -Name "hand_MinPosition_L" -SignalType "GO" -Device "Hand_L"\
      -Label "Min Position Left" -DeviceMap "16-23" -Category "HandLeft"\
      -Access "All" -Default 50

      -Name "hand_MaxSpeed_L" -SignalType "GO" -Device "Hand_L"\
      -Label "Max Speed Left" -DeviceMap "24-31" -Category "HandLeft"\
      -Access "All" -Default 200

      -Name "hand_HoldForce_L" -SignalType "GO" -Device "Hand_L"\
      -Label "Hold Force Left" -DeviceMap "40-47" -Category "HandLeft"\
      -Access "All" -Default 120

      -Name "hand_CmdVacuum1_L" -SignalType "DO" -Device "Hand_L"\
      -Label "Vacuum 1 Left" -DeviceMap "48" -Category "HandLeft" -Access "All"

      -Name "hand_CmdVacuum2_L" -SignalType "DO" -Device "Hand_L"\
      -Label "Vacuum 2 Left" -DeviceMap "49" -Category "HandLeft" -Access "All"

      -Name "hand_CmdBlowoff1_L" -SignalType "DO" -Device "Hand_L"\
      -Label "BlowOff 1 Left" -DeviceMap "50" -Category "HandLeft" -Access "All"

      -Name "hand_CmdBlowoff2_L" -SignalType "DO" -Device "Hand_L"\
      -Label "BlowOff 2 Left" -DeviceMap "51" -Category "HandLeft" -Access "All"

      -Name "hand_SysState_L" -SignalType "GI" -Device "Hand_L"\
      -Label "Finger State Left" -DeviceMap "0-4" -Category "HandLeft"\
      -Access "All"

      -Name "hand_SysError_L" -SignalType "GI" -Device "Hand_L"\
      -Label "Finger Error Left" -DeviceMap "32-39" -Category "HandLeft"\
      -Access "All"

      -Name "hand_StatusCalibrated_L" -SignalType "DI" -Device "Hand_L"\
      -Label "Calibrated Left" -DeviceMap "5" -Category "HandLeft" -Access "All"

      -Name "hand_ActualPosition_L" -SignalType "GI" -Device "Hand_L"\
      -Label "Actual Position Left" -DeviceMap "8-15" -Category "HandLeft"\
      -Access "All"

      -Name "hand_ActualSpeed_L" -SignalType "GI" -Device "Hand_L"\
      -Label "Actual Speed Left" -DeviceMap "16-23" -Category "HandLeft"\
      -Access "All"

      -Name "hand_StatusCamLinked_L" -SignalType "DI" -Device "Hand_L"\
      -Label "Camera Connection Left" -DeviceMap "40" -Category "HandLeft"\
      -Access "All"

      -Name "hand_SoftwareVersion_L" -SignalType "GI" -Device "Hand_L"\
      -Label "Software Version Left" -DeviceMap "41-47" -Category "HandLeft"\
      -Access "All"

      -Name "hand_StatusVacuum1_L" -SignalType "DI" -Device "Hand_L"\
      -Label "Vacuum 1 Left Status" -DeviceMap "48" -Category "HandLeft"\
      -Access "All"

      -Name "hand_StatusVacuum2_L" -SignalType "DI" -Device "Hand_L"\
      -Label "Vacuum 1 Left Status" -DeviceMap "49" -Category "HandLeft"\
      -Access "All"

      -Name "hand_StatusBlowoff1_L" -SignalType "DI" -Device "Hand_L"\
      -Label "SuncTool 1 Left Status" -DeviceMap "50" -Category "HandLeft"\
      -Access "All"

      -Name "hand_StatusBlowoff2_L" -SignalType "DI" -Device "Hand_L"\
      -Label "SuncTool 1 Left Status" -DeviceMap "51" -Category "HandLeft"\
      -Access "All"

      -Name "hand_ActualPressure1_L" -SignalType "GI" -Device "Hand_L"\
      -Label "Vacuum pressure1 Left" -DeviceMap "64-71" -Category "HandLeft"\
      -Access "All"

      -Name "hand_ActualPressure2_L" -SignalType "GI" -Device "Hand_L"\
      -Label "Vacuum pressure2 Left" -DeviceMap "72-79" -Category "HandLeft"\
      -Access "All"

      -Name "hand_SecurityKey_L" -SignalType "GO" -Device "Hand_L"\
      -Label "Security key Left" -DeviceMap "64-71" -Category "HandLeft"\
      -Access "All"

      -Name "hand_TftPFtpMode_L" -SignalType "DI" -Device "Hand_L"\
      -Label "Hand firmware update mode" -DeviceMap "7" -Category "HandLeft"\
      -Access "All"
